RoboDK station: robot_base.rdk

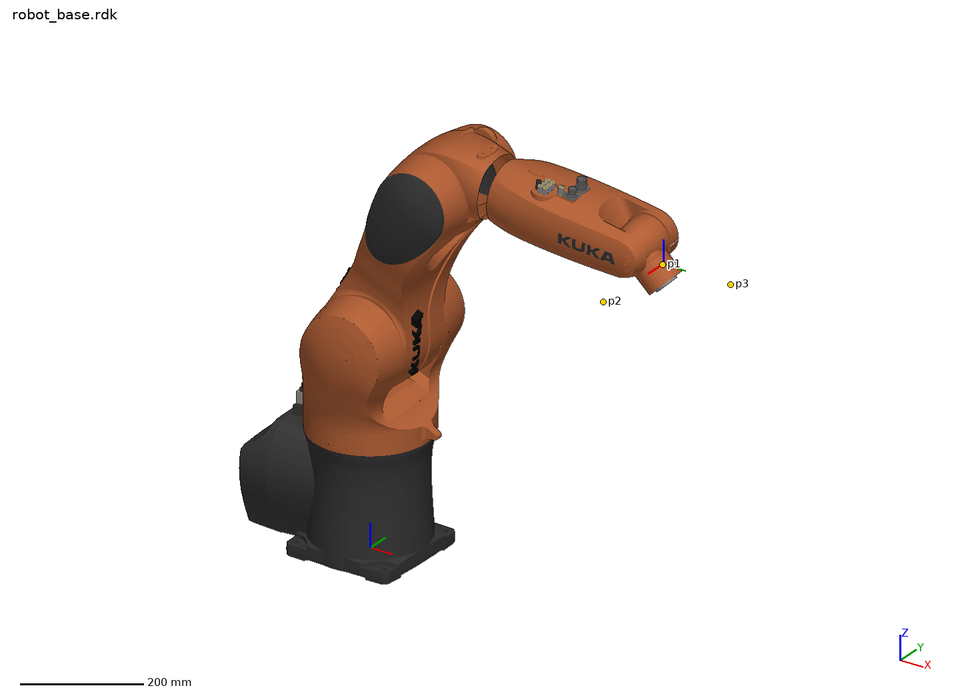
[picture v0: the station drawn from its stored meshes, robots at their saved joint values, targets as dots, program paths as lines]
Station robot_base (saved by RoboDK 5.3.0). Poses are relative to the parent item; angles as X-Y-Z fixed-axis rotations.
Station parameters (name, value as stored): $OUT[16], True
  - frame KUKA KR 6 R700 sixx Base at (0, 0, 0) mm
    - robot KUKA KR 6 R700 sixx: 6 axes, payload 6 kg, reach 706.7 mm, repeatability 0.03 mm, weight 50 kg
        modified DH rows (alpha deg, a mm, theta deg, d mm): 0, 0, 0, 400; -90, 25, 0, 0; 0, 315, -90, 0; -90, 35, 0, 365; 90, 0, 0, 0; -90, 0, 180, 80
        joint limits [-170, -190, -120, -185, -120, -350] to [170, 45, 156, 185, 120, 350]; home [0, -90, 90, 0, 0, 0]; saved at [-1.896, -66.969, 73.841, -2.462, 38.906, 5.559]
    - target p1 (joint target) at (520.93, 79.44, 622.96) mm, rotated rx -179.36 ry 45.86 rz -179.56 deg; joints [-9.78, -75.36, 84.92, 12.63, 35.7, -16.86] of KUKA KR 6 R700 sixx
    - target p2 (joint target) at (520.94, -88.29, 622.98) mm, rotated rx -179.36 ry 45.86 rz -179.57 deg; joints [10.73, -75.1, 84.6, -12.65, 35.76, 18.13] of KUKA KR 6 R700 sixx
    - target p3 (joint target) at (653.73, 82.08, 623.01) mm, rotated rx -179.36 ry 45.87 rz -179.57 deg; joints [-7.88, -47.37, 45.49, 8.23, 46.61, -10.88] of KUKA KR 6 R700 sixx
    - frame task_frame at (520.93, 82.08, 622.96) mm, rotated rx 0.02 ry -0.01 rz -90 deg
  - Python program 3Dprint_offline (listed below)

--- Python program 3Dprint_offline ---
# Type help("robolink") or help("robodk") for more information
# Documentation: https://robodk.com/doc/en/RoboDK-API.html
# Reference:     https://robodk.com/doc/en/PythonAPI/index.html
# Note: It is not required to keep a copy of this file, your python script is saved with the station
from robolink import *                                              # RoboDK API
from robodk import *                                                # Robot toolbox
import time                                                         # Standard time library
import re                                                           # Imports the regex expressions

######################################################### FUNCTIONS #########################################################


def extruder_offline(robot, arg):
    '''Turns on and off the extrusion '''                           # Not used in code for reasons described above
    if arg == 'START':                                              # User sets the arg to start printing
        robot.setDO('$OUT[16]', 'True')                             # Set the output value to start printing
    elif arg == 'STOP':                                             # User sets the arg to stop printing
        robot.setDO('$OUT[16]', 'False')                            # Set the output value to stop printing
    else:
        print('The input of extruder() has to be either START or STOP')

def parser(filename):
    '''Parse gcode commands to be used in our code'''
    parsed_file = list()                                            # Create a list
    layer = 0                                                       # Z-axis, or current height of the print
    with open(filename) as gcode:                                   # Open gcode path and use as variable
        for line in gcode:                                          # For each line in gcode:
            line = line.strip()                                     # Delete all unnecessary ASCII characters
            if re.findall("LAYER:", line):                          # If new layer found, update z-axes
                layer += 1                                          # Add the layer value
                continue                                            # Skip the next if
            if re.findall("G1", line):                              # Check if line begins with "G1"
                coord = re.findall(r'[XY].?\d+.\d+', line)          # Assign coord values
                if len(coord) == 2:                                 # If both coords were assigned
                    X = re.findall('\d*\.?\d+', coord[0])[0]        # Assign X-value
                    Y = re.findall('\d*\.?\d+', coord[1])[0]        # Assign Y-value
                    parsed_file.append([float(X), float(Y), layer, True])   # Append our desired output for use in the project
    return parsed_file


########################################################### MAIN ###########################################################

# ROBODK INITIALIZATION
RDK = Robolink()                                                     # sys.path.insert(0, "C:\ProgramFiles\RoboDK\Python")
robot = RDK.Item('KUKA KR 6 R700 sixx')                              # Create the robot instance
RDK.setSimulationSpeed(1)                                            # ADJUSTABLE: Simulation speed (1=default)
reference = robot.Parent()                                           # Retrieve the robot reference frame
robot.setPoseFrame(reference)                                        # Use the robot base frame as active reference
home = [0, -90, 90, 0, 0, 0]                                         # Setup the home joint position
robot.MoveJ(home)                                                    # Move to home in RoboDK
robot.setSpeed(speed_linear=100)                                     # ADJUSTABLE: Change the printing speed here
layer_height = 0.55                                                  # ADJUSTABLE: edit the layer height
path = parser('desired/path/to/gcode') # ADJUSTABLE: Parse the gcode
item_frame = RDK.Item('task_frame')                                  # ADJUSTABLE Load the task_frame from RoboDK
home_joints = [-5.520000, -107.550000, 115.910000, 1.620000,
               37.390000, -0.2400006]                                # ADJUSTABLE Orient robot with joints to P1
robot.setFrame(item_frame)                                           # Set the robot frame
robot.MoveJ(home_joints)                                             # Move to home position (First move must be in joints)


# TOOL ORIENTATION + INVERSE KINEMATICS
orient_frame2tool = invH(item_frame.Pose())*robot.SolveFK(home_joints)  # Homogeneous matrix * joint orientation
orient_frame2tool[0:3, 3] = Mat([0, 0, 0])                              # Remove the last column of homogeneous matrix


# TASK_FRAME CHECK
robot.MoveL(transl([0, 0, 0])*orient_frame2tool)                      # Move to the first corner
robot.MoveL(transl([0, 70, 0])*orient_frame2tool)                     # Move to the second corner
robot.MoveL(transl([70, 70, 0])*orient_frame2tool)                    # Move to the third corner
robot.MoveL(transl([70, 0, 0])*orient_frame2tool)                     # Move to the forth corner
robot.MoveL(transl([0, 0, 0])*orient_frame2tool)                      # Move back to the start


# GET RID OF EXTRA FILAMENT (CAN BE REMOVED)
robot.MoveL(transl([0, 0, 0])*orient_frame2tool)                      # Printing blob
time.sleep(2)                                                         # Used to leave the blob
robot.MoveL(transl([0, 0, 3])*orient_frame2tool)                      # Move up to get rid of the filament


# PRINTING
RDK.setSimulationSpeed(1)                                             # ADJUSTABLE, set to default speed
printing_status = False                                               # Default value for printing status
for item in path:                                                     # Go through each coordinate from the parsed GCode file
    if item[3] == False and printing_status == True:                  # If we want to stop extrusion which is running right now
        extruder_offline(robot, "STOP")                               # Function to stop extrusion is called
        printing_status = False                                       # Set the printing status to false
    elif item[3] == True and printing_status == False:                # If we want to start printing and we are not
        extruder_offline(robot, "START")                              # Call the function to start extruding
        printing_status = True                                        # Set the printing status to true
    target_point = [item[0], item[1], layer_height*item[2]+0.15]      # ADJSUTABLE, call the coord to go to, 0.55 is the layer heigh
    target0 = transl(target_point)*orient_frame2tool                  # Set the target point with correct rotation of the extruder
    robot.MoveL(target0, blocking=False)                              # Move the robot to target
robot.MoveJ(home)                                                     # Move back home at the end of program
